{attribute 'linkalways'} 
{attribute 'no_explicit_call' := 'This FB is a CLASS and must be accessed using methods or properties'}
{attribute 'enable_dynamic_creation'}
FUNCTION_BLOCK FINAL GT_REAL EXTENDS Node
VAR
	in1 : _REAL(0.0);
	in2 : _REAL(0.0);
	out : _BOOL(FALSE);
END_VAR

METHOD PUBLIC Clone : I_Node
VAR
	pNode : POINTER TO GT_REAL;
END_VAR
pNode := __NEW(GT_REAL);
Clone := pNode^;
END_METHOD

METHOD FB_init : BOOL
VAR_INPUT
	bInitRetains : BOOL; // if TRUE, the retain variables are initialized (warm start / cold start)
	bInCopyCode : BOOL;  // if TRUE, the instance afterwards gets moved into the copy code (online change)
END_VAR
AddInput('in1',THIS^.in1);
AddInput('in2',THIS^.in2);
AddOutput('out', THIS^.out);
END_METHOD

METHOD PROTECTED OnExecute
VAR
END_VAR
out.Value := in1.Value > in2.Value;
END_METHOD

END_FUNCTION_BLOCK

(* stored: Version 1.1.0.1, ProductVersion 3.1.4024.15
   POU GT_REAL: Id {a0a7a50f-0eda-4755-b772-a086ad5267af}, SpecialFunc None
   Folder Constructor: Id {ff782e8e-c30a-4bed-b210-5c419cb05689}
   Method Clone: Id {7d060c31-cd29-4779-a049-4cdfb05cdb53}
   Method FB_init: Id {32225ef8-50da-42a9-82be-e27359ec1359}
   Method OnExecute: Id {3ad53dbd-b030-4d2e-a7d5-dcaaf0b28c72} *)
